{attribute 'GeneratedUsingTerminal: AT2025-0250-0022'}
{attribute addProperty BoxType "AT2025-0250-0022"}
{attribute addProperty Id "A_0075_AT2000_5250_0019_AT2000_5250AT2000_01D6DEDF80"}
{attribute addProperty CRC "2047902286"}
{attribute addProperty Size "80"}
TYPE A_0063_AT2025_0250_0022_AT2025_0250_7A10824E EXTENDS AT2025_86175B41 :
STRUCT
	{attribute addProperty Name "A_0075_AT2000_5250_0019_AT2000_5250"}
	{attribute addProperty PreviousPort "A_0063(AT2025-0250-0022) (AT2025-0250) : B"}
	A_0075_AT2000_5250_0019_AT2000_5250 : AT2000_01D6DEDF;
END_STRUCT
END_TYPE

(* stored: Version 1.2.0.0, ProductVersion 3.1.4024.9
   DUT A_0063_AT2025_0250_0022_AT2025_0250_7A10824E: Id {f2adf5f8-23e7-4c2f-ab6b-59291c1c8914} *)
